TYPE "MEStoPLC_MainCheckOut_ext"
VERSION : 0.1
   STRUCT
      UnloadLoad_ResultsStored1OK : Bool;
      UnloadLoad_ResultsStored1NG : Bool;
      UnloadLoad_ResultsStored1ReqMesDone : Bool;
      UnloadLoad_ResultsStored1Spare : Bool;
      UnloadLoad_ResultsStored1Spare1 : Bool;
      UnloadLoad_ResultsStored1Spare2 : Bool;
      UnloadLoad_ResultsStored1Spare3 : Bool;
      UnloadLoad_ResultsStored1Spare4 : Bool;
      UnloadLoad_ResultsStored2OK : Bool;
      UnloadLoad_ResultsStored2NG : Bool;
      UnloadLoad_ResultsStored2ReqMesDone : Bool;
      UnloadLoad_ResultsStored2Spare : Bool;
      UnloadLoad_ResultsStored2Spare1 : Bool;
      UnloadLoad_ResultsStored2Spare2 : Bool;
      UnloadLoad_ResultsStored2Spare3 : Bool;
      UnloadLoad_ResultsStored2Spare4 : Bool;
      UnloadLoad_ResultsStored3OK : Bool;
      UnloadLoad_ResultsStored3NG : Bool;
      UnloadLoad_ResultsStored3ReqMesDone : Bool;
      UnloadLoad_ResultsStored3Spare : Bool;
      UnloadLoad_ResultsStored3Spare1 : Bool;
      UnloadLoad_ResultsStored3Spare2 : Bool;
      UnloadLoad_ResultsStored3Spare3 : Bool;
      UnloadLoad_ResultsStored3Spare4 : Bool;
      UnloadLoad_ResultsStored4OK : Bool;
      UnloadLoad_ResultsStored4NG : Bool;
      UnloadLoad_ResultsStored4ReqMesDone : Bool;
      UnloadLoad_ResultsStored4Spare : Bool;
      UnloadLoad_ResultsStored4Spare1 : Bool;
      UnloadLoad_ResultsStored4Spare2 : Bool;
      UnloadLoad_ResultsStored4Spare3 : Bool;
      UnloadLoad_ResultsStored4Spare4 : Bool;
      UnloadLoad_ResultsStored5OK : Bool;
      UnloadLoad_ResultsStored5NG : Bool;
      UnloadLoad_ResultsStored5ReqMesDone : Bool;
      UnloadLoad_ResultsStored5Spare : Bool;
      UnloadLoad_ResultsStored5Spare1 : Bool;
      UnloadLoad_ResultsStored5Spare2 : Bool;
      UnloadLoad_ResultsStored5Spare3 : Bool;
      UnloadLoad_ResultsStored5Spare4 : Bool;
      UnloadLoad_ResultsStored6OK : Bool;
      UnloadLoad_ResultsStored6NG : Bool;
      UnloadLoad_ResultsStored6ReqMesDone : Bool;
      UnloadLoad_ResultsStored6Spare : Bool;
      UnloadLoad_ResultsStored6Spare1 : Bool;
      UnloadLoad_ResultsStored6Spare2 : Bool;
      UnloadLoad_ResultsStored6Spare3 : Bool;
      UnloadLoad_ResultsStored6Spare4 : Bool;
      UnloadLoad_ResultsStored7OK : Bool;
      UnloadLoad_ResultsStored7NG : Bool;
      UnloadLoad_ResultsStored7ReqMesDone : Bool;
      UnloadLoad_ResultsStored7Spare : Bool;
      UnloadLoad_ResultsStored7Spare1 : Bool;
      UnloadLoad_ResultsStored7Spare2 : Bool;
      UnloadLoad_ResultsStored7Spare3 : Bool;
      UnloadLoad_ResultsStored7Spare4 : Bool;
      UnloadLoad_ResultsStored8OK : Bool;
      UnloadLoad_ResultsStored8NG : Bool;
      UnloadLoad_ResultsStored8ReqMesDone : Bool;
      UnloadLoad_ResultsStored8Spare : Bool;
      UnloadLoad_ResultsStored8Spare5 : Bool;
      UnloadLoad_ResultsStored8Spare6 : Bool;
      UnloadLoad_ResultsStored8Spare8 : Bool;
      UnloadLoad_ResultsStored8Spare9 : Bool;
   END_STRUCT;

END_TYPE

